TEXTLIST AnyStationWarningList
  0 = ' '
  1 = 'Station 1 Warn'
  2 = 'Station 2 Warn'
  3 = 'Station 3 Warn'
  4 = 'Station 4 Warn'
  5 = 'Station 5 Warn'
  6 = 'Station 6 Warn'
  99 = 'Machine Warn'
   = ''
END_TEXTLIST

(* stored: Version 1.1.0.1, ProductVersion 3.1.4024.12
   TextList AnyStationWarningList: Id {fa236f4e-9fc4-4f59-88ec-cdc064d685a6} *)
